# EPICS autosave request: dxp/tags/R3-5/dxpApp/Db/dxpMapping_settings.req
$(P)CollectMode
$(P)ListMode
$(P)PixelAdvanceMode
$(P)PixelsPerRun
$(P)AutoPixelsPerBuffer
$(P)PixelsPerBuffer
$(P)IgnoreGate
$(P)SyncCount
$(P)InputLogicPolarity
